// Mitsubishi GX Works2 project: EX2_20 (1)   PLC: FX3G

// global labels: Global1
VAR_GLOBAL CONSTANT
  Reset_analog : REAL;
END_VAR
VAR_GLOBAL
  Starter AT X007 : BOOL;
  Emergency AT X005 : BOOL;
  Workday_Lamp AT Y007 : BOOL;
END_VAR
VAR_GLOBAL CONSTANT
  Const_400 : REAL := 400;
  Const_100 : REAL := 100;
  Const_120 : REAL := 120;
  Const_60 : REAL := 60;
  Reset : INT;
END_VAR
VAR_GLOBAL
  Start_Melt AT X001 : BOOL;
  Analog_Input1 AT D8280 : INT;
  Invert_analog_Input1 AT D1170 : REAL;
  Start_fill AT X004 : BOOL;
END_VAR
VAR_GLOBAL CONSTANT
  Convert_input : REAL := 400.0;
END_VAR
VAR_GLOBAL
  New_analog_input2 AT D1160 : REAL;
  begin_analog_input AT M1 : BOOL;
  Analog_Output AT D8282 : INT;
  Choco_Input AT D1110 : REAL;
  Nut_Input AT D1120 : REAL;
  Fistuk_Input AT D1130 : REAL;
  Kadaif_Input AT D1140 : REAL;
  Choco_Stock AT D1210 : REAL;
  Nut_Stock AT D1220 : REAL;
  Fistuk_Stock AT D1230 : REAL;
  Kadaif_Stock AT D1240 : REAL;
  Invalid_out AT M10 : BOOL;
  begin_analog1 AT M1 : BOOL;
  active_melt AT Y001 : BOOL;
  temp_sensor AT X002 : BOOL;
END_VAR
VAR_GLOBAL CONSTANT
  Choco_to_melt : REAL := 400;
END_VAR
VAR_GLOBAL
  location_sensor AT X003 : BOOL;
  Cast_lamp AT Y002 : BOOL;
  Casting AT TS2 : BOOL;
END_VAR
VAR_GLOBAL CONSTANT
  casting_time : INT := 40;
END_VAR
VAR_GLOBAL
  t_cast AT TC2 : BOOL;
  Melt_finished AT M4 : BOOL;
  End_day AT M9 : BOOL;
END_VAR
VAR_GLOBAL CONSTANT
  Const_5 : REAL := 5;
END_VAR
VAR_GLOBAL
  final_analog_input1 AT D1160 : REAL;
  Nuts_cream AT M2 : BOOL;
  Dubai_cream AT M5 : BOOL;
END_VAR
VAR_GLOBAL CONSTANT
  Const_20 : REAL := 20;
END_VAR
VAR_GLOBAL
  Cream_end AT M3 : BOOL;
  Mix_Container AT D1180 : REAL;
END_VAR
VAR_GLOBAL CONSTANT
  Const_200 : REAL := 200;
END_VAR
VAR_GLOBAL
  timer3 AT TC3 : BOOL;
END_VAR
VAR_GLOBAL CONSTANT
  filling_time : INT := 25;
END_VAR
VAR_GLOBAL
  timer4 AT TC4 : BOOL;
  flash_lightA AT TS3 : BOOL;
  flash_control AT M20 : BOOL;
  flashA AT Y003 : BOOL;
  flash_lightB AT TS4 : BOOL;
  flashB AT Y004 : BOOL;
  Start_Cold AT X006 : BOOL;
  Colding AT TS5 : BOOL;
  Colding_lamp AT Y006 : BOOL;
  t_cold AT TC5 : BOOL;
END_VAR
VAR_GLOBAL CONSTANT
  colding_time : INT := 30;
END_VAR
VAR_GLOBAL
  finish_cold AT M6 : BOOL;
  timer1 AT TC1 : BOOL;
END_VAR
VAR_GLOBAL CONSTANT
  Total_filling : INT := 50;
END_VAR
VAR_GLOBAL
  total_fill AT TS1 : BOOL;
  Packing_lamp AT Y005 : BOOL;
END_VAR
VAR_GLOBAL CONSTANT
  pack_target : INT := 4;
END_VAR
VAR_GLOBAL
  Counter1 AT CC2 : BOOL;
  Pack_chocolate AT X000 : BOOL;
  done_packing AT M7 : BOOL;
  CS2_out AT CS2 : BOOL;
END_VAR
VAR_GLOBAL CONSTANT
  Const_4 : REAL := 4;
END_VAR
VAR_GLOBAL
  Ready_Chocolate AT D1290 : REAL;
END_VAR
VAR_GLOBAL CONSTANT
  Const_1 : REAL := 1;
END_VAR
VAR_GLOBAL
  Num_Packs AT D1300 : REAL;
END_VAR
VAR_GLOBAL CONSTANT
  Reset_float : REAL;
  Reset_bit : BOOL;
  Const_10 : REAL := 10.0;
  Const_40 : INT := 40;
END_VAR
VAR_GLOBAL
  Packs_Storage AT D3000 : REAL;
END_VAR
VAR_GLOBAL CONSTANT
  Const_01 : REAL := 0.1;
END_VAR

// task Task_01 (event TRUE, interval 0, priority 31): POU_01

PROGRAM POU_01
(* structured ladder/FBD written out as ST: instructions are called as NAME(EN, inputs, outputs); _pN, _eN, _tN stand for wires *)
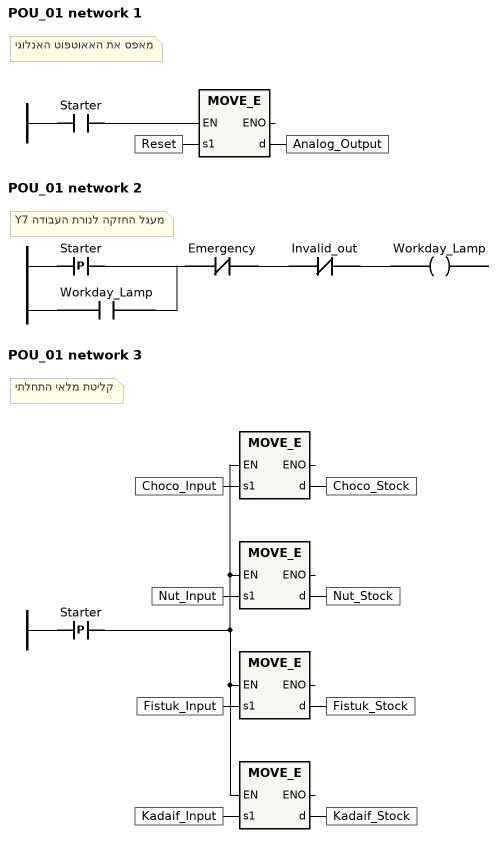
(* network 1 *)
(* מאפס את האאוטפוט האנלוגי *)
MOVE_E(Starter, Reset, Analog_Output);
(* network 2 *)
(* מעגל החזקה לנורת העבודה Y7 *)
Workday_Lamp := ((LDP(TRUE, Starter) OR Workday_Lamp) AND NOT Emergency) AND NOT Invalid_out;
(* network 3 *)
(* קליטת מלאי התחלתי *)
_p1 := LDP(TRUE, Starter);
MOVE_E(_p1, Choco_Input, Choco_Stock);
MOVE_E(_p1, Nut_Input, Nut_Stock);
MOVE_E(_p1, Fistuk_Input, Fistuk_Stock);
MOVE_E(_p1, Kadaif_Input, Kadaif_Stock);
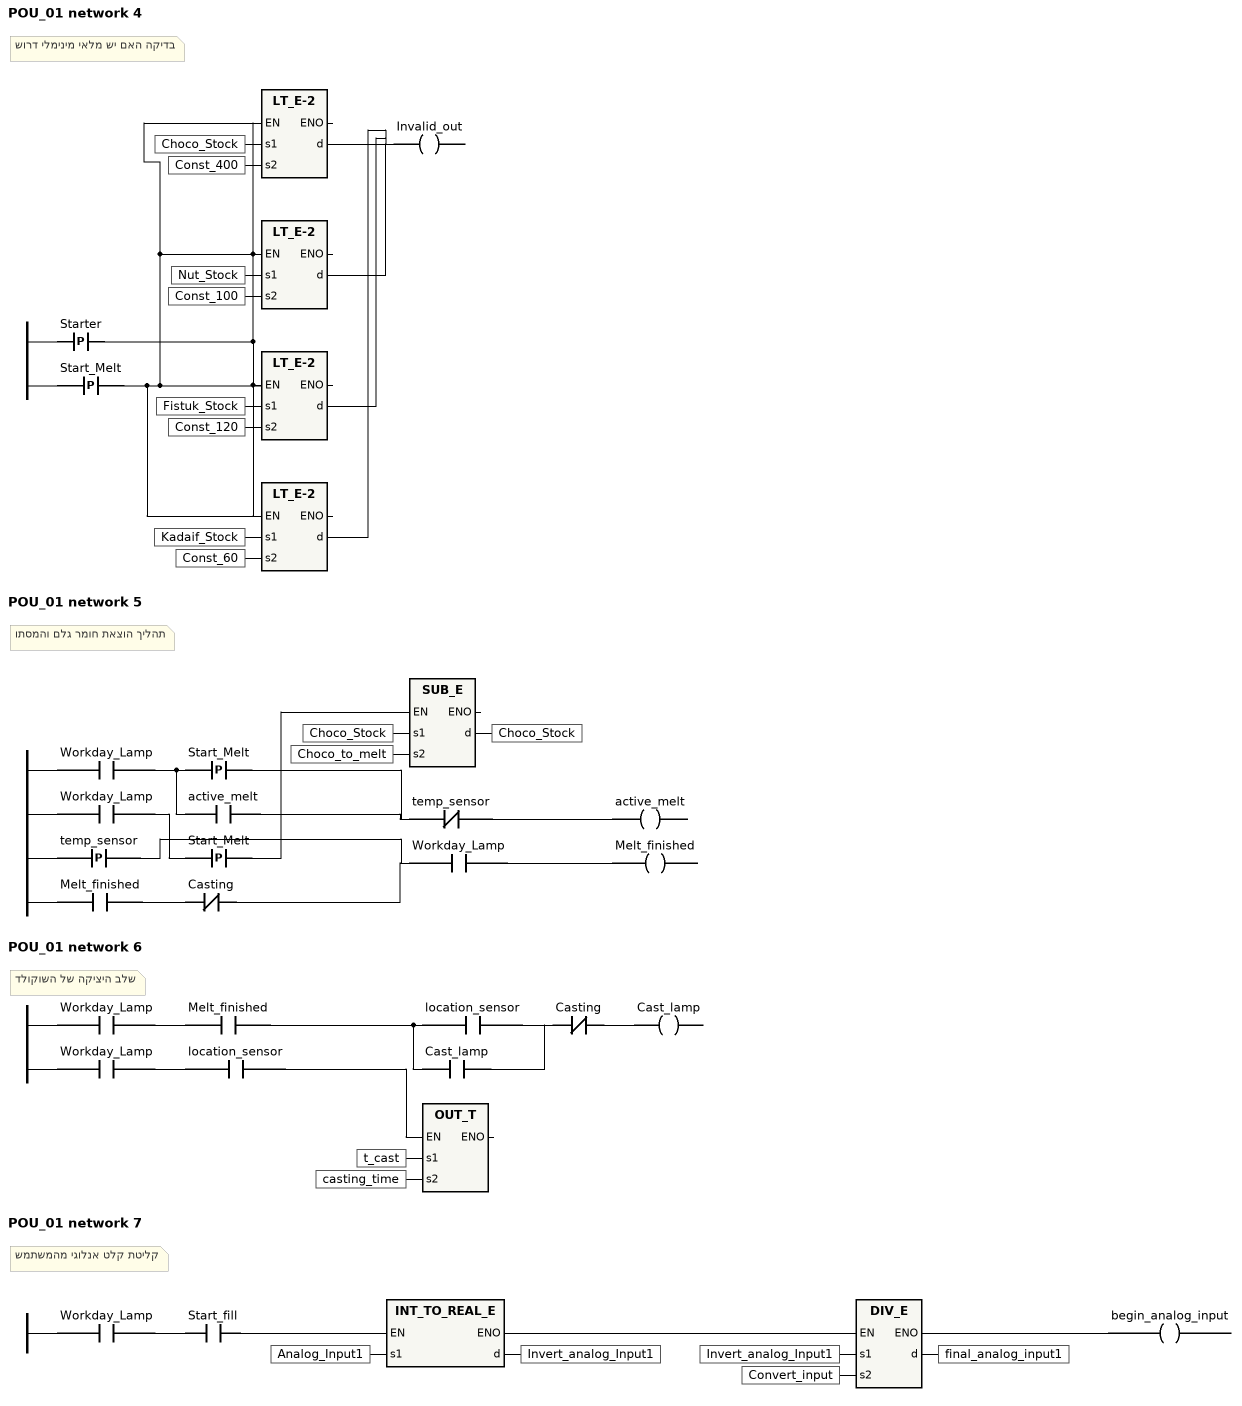
(* network 4 *)
(* בדיקה האם יש מלאי מינימלי דרוש *)
_p1 := LDP(TRUE, Starter) OR LDP(TRUE, Start_Melt);
LT_E(_p1, Choco_Stock, Const_400, _t2);
LT_E(_p1, Nut_Stock, Const_100, _t3);
LT_E(_p1, Fistuk_Stock, Const_120, _t4);
LT_E(_p1, Kadaif_Stock, Const_60, _t5);
Invalid_out := _t2 OR _t3 OR _t4 OR _t5;
(* network 5 *)
(* תהליך הוצאת חומר גלם והמסתו *)
active_melt := ((Workday_Lamp AND LDP(TRUE, Start_Melt)) OR (Workday_Lamp AND active_melt)) AND NOT temp_sensor;
SUB_E(Workday_Lamp AND LDP(TRUE, Start_Melt), Choco_Stock, Choco_to_melt, Choco_Stock);
Melt_finished := (LDP(TRUE, temp_sensor) OR (Melt_finished AND NOT Casting)) AND Workday_Lamp;
(* network 6 *)
(* שלב היציקה של השוקולד *)
_p1 := Workday_Lamp AND Melt_finished;
Cast_lamp := ((_p1 AND location_sensor) OR (_p1 AND Cast_lamp)) AND NOT Casting;
OUT_T(Workday_Lamp AND location_sensor, t_cast, casting_time);
(* network 7 *)
(* קליטת קלט אנלוגי מהמשתמש *)
_e1 := INT_TO_REAL_E(Workday_Lamp AND Start_fill, Analog_Input1, Invert_analog_Input1);
_e2 := DIV_E(_e1, Invert_analog_Input1, Convert_input, final_analog_input1);
begin_analog_input := _e2;
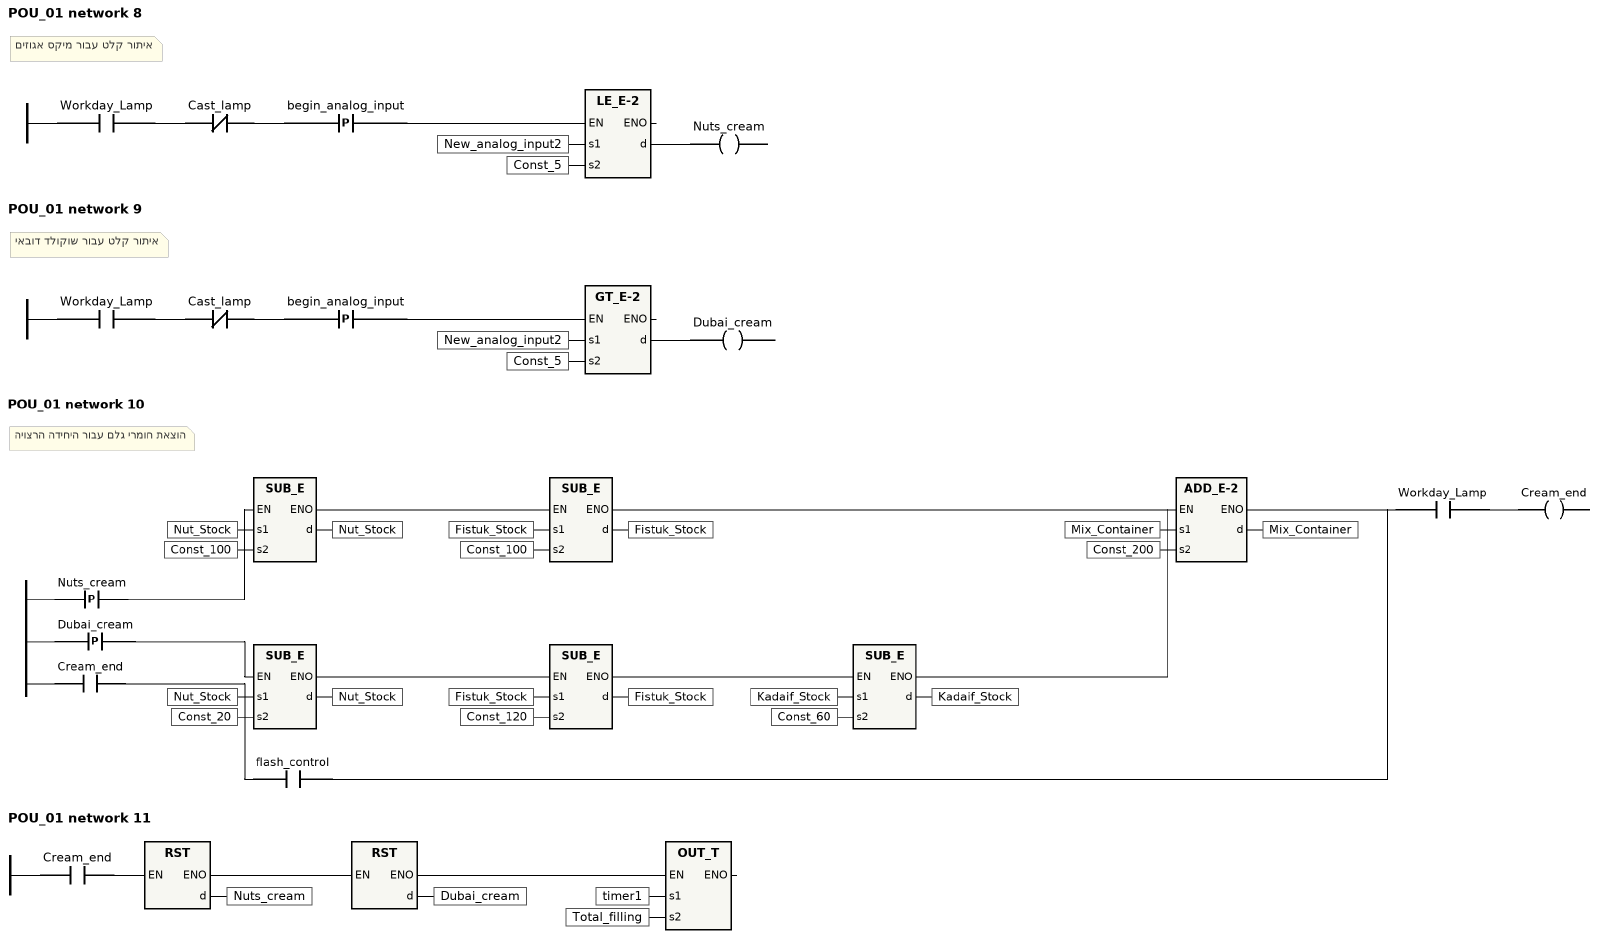
(* network 8 *)
(* איתור קלט עבור מיקס אגוזים *)
LE_E(Workday_Lamp AND NOT Cast_lamp AND LDP(TRUE, begin_analog_input), New_analog_input2, Const_5, _t1);
Nuts_cream := _t1;
(* network 9 *)
(* איתור קלט עבור שוקולד דובאי *)
GT_E(Workday_Lamp AND NOT Cast_lamp AND LDP(TRUE, begin_analog_input), New_analog_input2, Const_5, _t1);
Dubai_cream := _t1;
(* network 10 *)
(* הוצאת חומרי גלם עבור היחידה הרצויה *)
_e1 := SUB_E(LDP(TRUE, Nuts_cream), Nut_Stock, Const_100, Nut_Stock);
_e2 := SUB_E(_e1, Fistuk_Stock, Const_100, Fistuk_Stock);
_e3 := SUB_E(LDP(TRUE, Dubai_cream), Nut_Stock, Const_20, Nut_Stock);
_e4 := SUB_E(_e3, Fistuk_Stock, Const_120, Fistuk_Stock);
_e5 := SUB_E(_e4, Kadaif_Stock, Const_60, Kadaif_Stock);
_e6 := ADD_E(_e2 OR _e5, Mix_Container, Const_200, Mix_Container);
Cream_end := (_e6 OR (Cream_end AND flash_control)) AND Workday_Lamp;
(* network 11 *)
_e1 := RST(Cream_end, Nuts_cream);
_e2 := RST(_e1, Dubai_cream);
OUT_T(_e2, timer1, Total_filling);
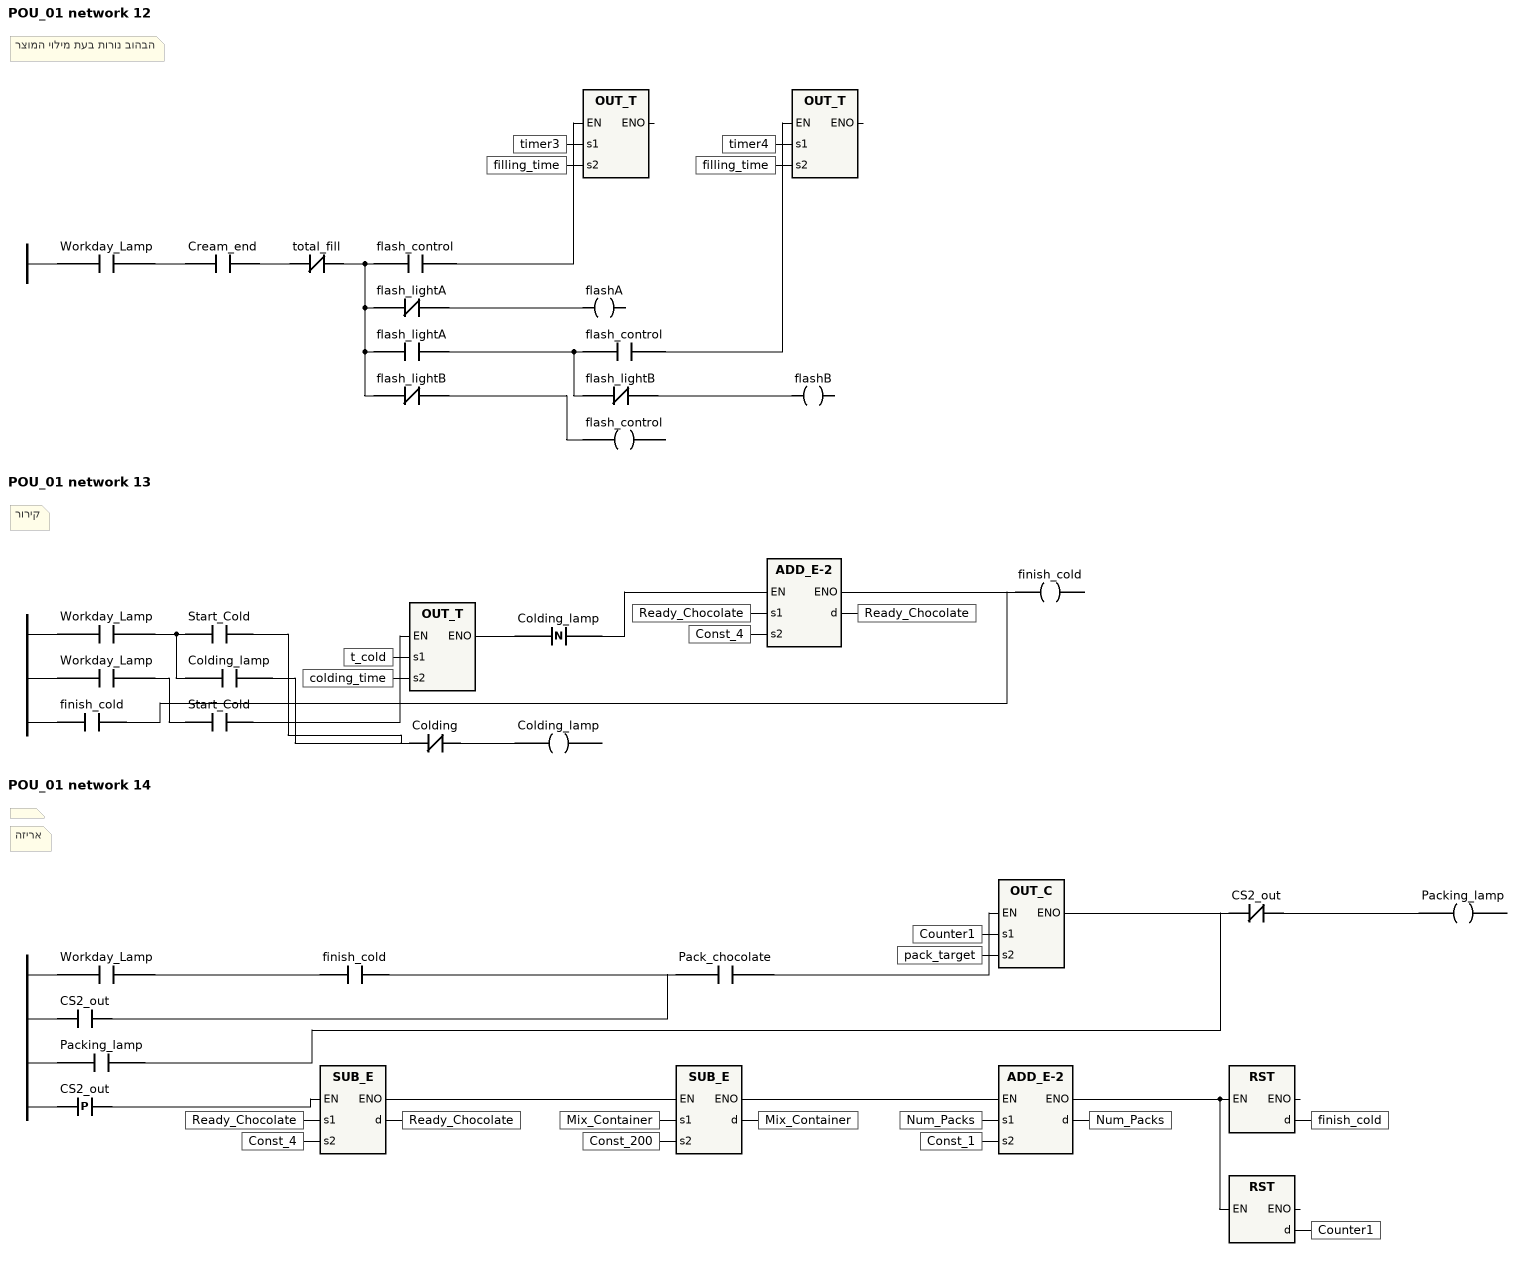
(* network 12 *)
(* הבהוב נורות בעת מילוי המוצר *)
_p1 := Workday_Lamp AND Cream_end AND NOT total_fill;
OUT_T(_p1 AND flash_control, timer3, filling_time);
flashA := _p1 AND NOT flash_lightA;
_p2 := _p1 AND flash_lightA;
OUT_T(_p2 AND flash_control, timer4, filling_time);
flashB := _p2 AND NOT flash_lightB;
flash_control := _p1 AND NOT flash_lightB;
(* network 13 *)
(* קירור *)
Colding_lamp := ((Workday_Lamp AND Start_Cold) OR (Workday_Lamp AND Colding_lamp)) AND NOT Colding;
_e1 := OUT_T(Workday_Lamp AND Start_Cold, t_cold, colding_time);
_e2 := ADD_E(_e1 AND LDF(TRUE, Colding_lamp), Ready_Chocolate, Const_4, Ready_Chocolate);
finish_cold := _e2 OR finish_cold;
(* network 14 *)
(*  *)
(* אריזה *)
_e1 := OUT_C(((Workday_Lamp AND finish_cold) OR CS2_out) AND Pack_chocolate, Counter1, pack_target);
Packing_lamp := (_e1 OR Packing_lamp) AND NOT CS2_out;
_e2 := SUB_E(LDP(TRUE, CS2_out), Ready_Chocolate, Const_4, Ready_Chocolate);
_e3 := SUB_E(_e2, Mix_Container, Const_200, Mix_Container);
_e4 := ADD_E(_e3, Num_Packs, Const_1, Num_Packs);
RST(_e4, finish_cold);
RST(_e4, Counter1);
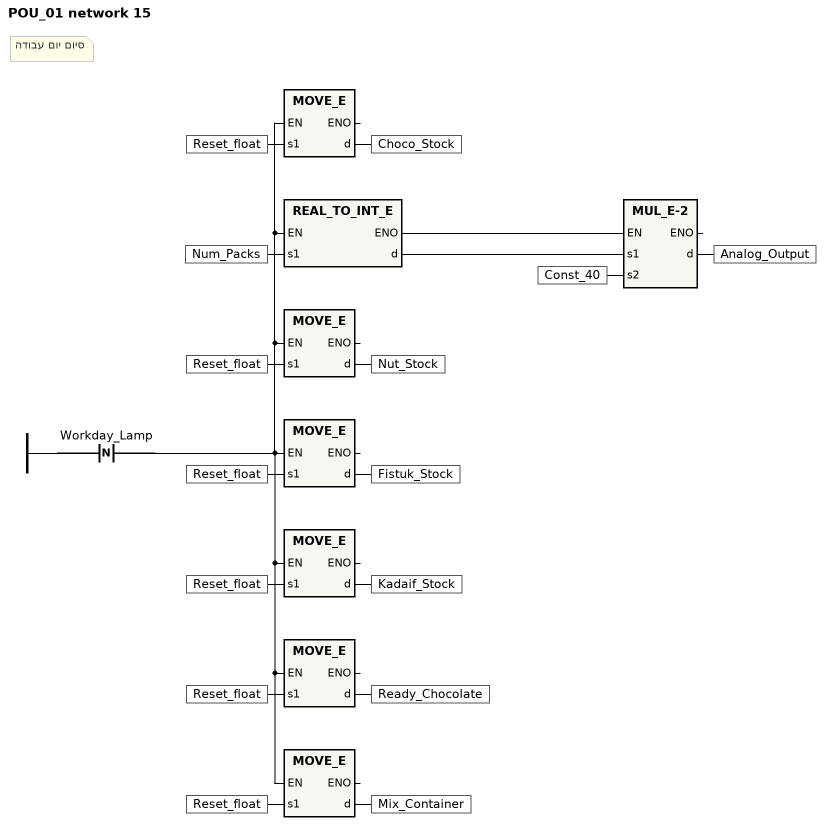
(* network 15 *)
(* סיום יום עבודה *)
_p1 := LDF(TRUE, Workday_Lamp);
MOVE_E(_p1, Reset_float, Choco_Stock);
MOVE_E(_p1, Reset_float, Nut_Stock);
MOVE_E(_p1, Reset_float, Fistuk_Stock);
MOVE_E(_p1, Reset_float, Kadaif_Stock);
MOVE_E(_p1, Reset_float, Ready_Chocolate);
MOVE_E(_p1, Reset_float, Mix_Container);
_e3 := REAL_TO_INT_E(_p1, Num_Packs, _t2);
MUL_E(_e3, _t2, Const_40, Analog_Output);
END_PROGRAM
